FUNCTION_BLOCK UA_UnitMux (* Serialises OPC UA method calls onto command events and routes the accept/reject answer back to the calling method's RSP *)
  (* Standard: 61499-2 *)
  (* Version 2.0, 2026-09-27, Project contributors, Filling cell reference model *)
  PACKAGE fillingcell;
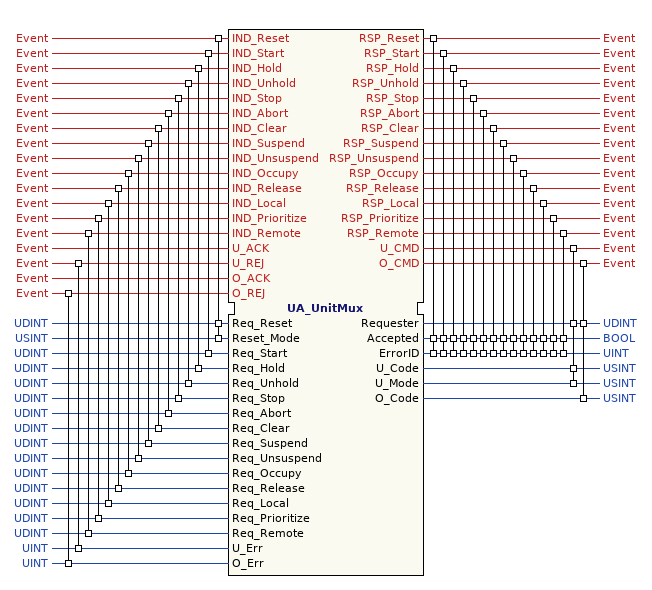
  EVENT_INPUT
    IND_Reset WITH Req_Reset, Reset_Mode;
    IND_Start WITH Req_Start;
    IND_Hold WITH Req_Hold;
    IND_Unhold WITH Req_Unhold;
    IND_Stop WITH Req_Stop;
    IND_Abort WITH Req_Abort;
    IND_Clear WITH Req_Clear;
    IND_Suspend WITH Req_Suspend;
    IND_Unsuspend WITH Req_Unsuspend;
    IND_Occupy WITH Req_Occupy;
    IND_Release WITH Req_Release;
    IND_Local WITH Req_Local;
    IND_Prioritize WITH Req_Prioritize;
    IND_Remote WITH Req_Remote;
    U_ACK;
    U_REJ WITH U_Err;
    O_ACK;
    O_REJ WITH O_Err;
  END_EVENT
  EVENT_OUTPUT
    RSP_Reset WITH Accepted, ErrorID;
    RSP_Start WITH Accepted, ErrorID;
    RSP_Hold WITH Accepted, ErrorID;
    RSP_Unhold WITH Accepted, ErrorID;
    RSP_Stop WITH Accepted, ErrorID;
    RSP_Abort WITH Accepted, ErrorID;
    RSP_Clear WITH Accepted, ErrorID;
    RSP_Suspend WITH Accepted, ErrorID;
    RSP_Unsuspend WITH Accepted, ErrorID;
    RSP_Occupy WITH Accepted, ErrorID;
    RSP_Release WITH Accepted, ErrorID;
    RSP_Local WITH Accepted, ErrorID;
    RSP_Prioritize WITH Accepted, ErrorID;
    RSP_Remote WITH Accepted, ErrorID;
    U_CMD WITH Requester, U_Code, U_Mode;
    O_CMD WITH Requester, O_Code;
  END_EVENT
  VAR_INPUT
    Req_Reset : UDINT;
    Reset_Mode : USINT;
    Req_Start : UDINT;
    Req_Hold : UDINT;
    Req_Unhold : UDINT;
    Req_Stop : UDINT;
    Req_Abort : UDINT;
    Req_Clear : UDINT;
    Req_Suspend : UDINT;
    Req_Unsuspend : UDINT;
    Req_Occupy : UDINT;
    Req_Release : UDINT;
    Req_Local : UDINT;
    Req_Prioritize : UDINT;
    Req_Remote : UDINT;
    U_Err : UINT := 5;
    O_Err : UINT := 5;
  END_VAR
  VAR_OUTPUT
    Requester : UDINT;
    Accepted : BOOL;
    ErrorID : UINT;
    U_Code : USINT;
    U_Mode : USINT;
    O_Code : USINT;
  END_VAR
  VAR
    Pending : USINT;
  END_VAR
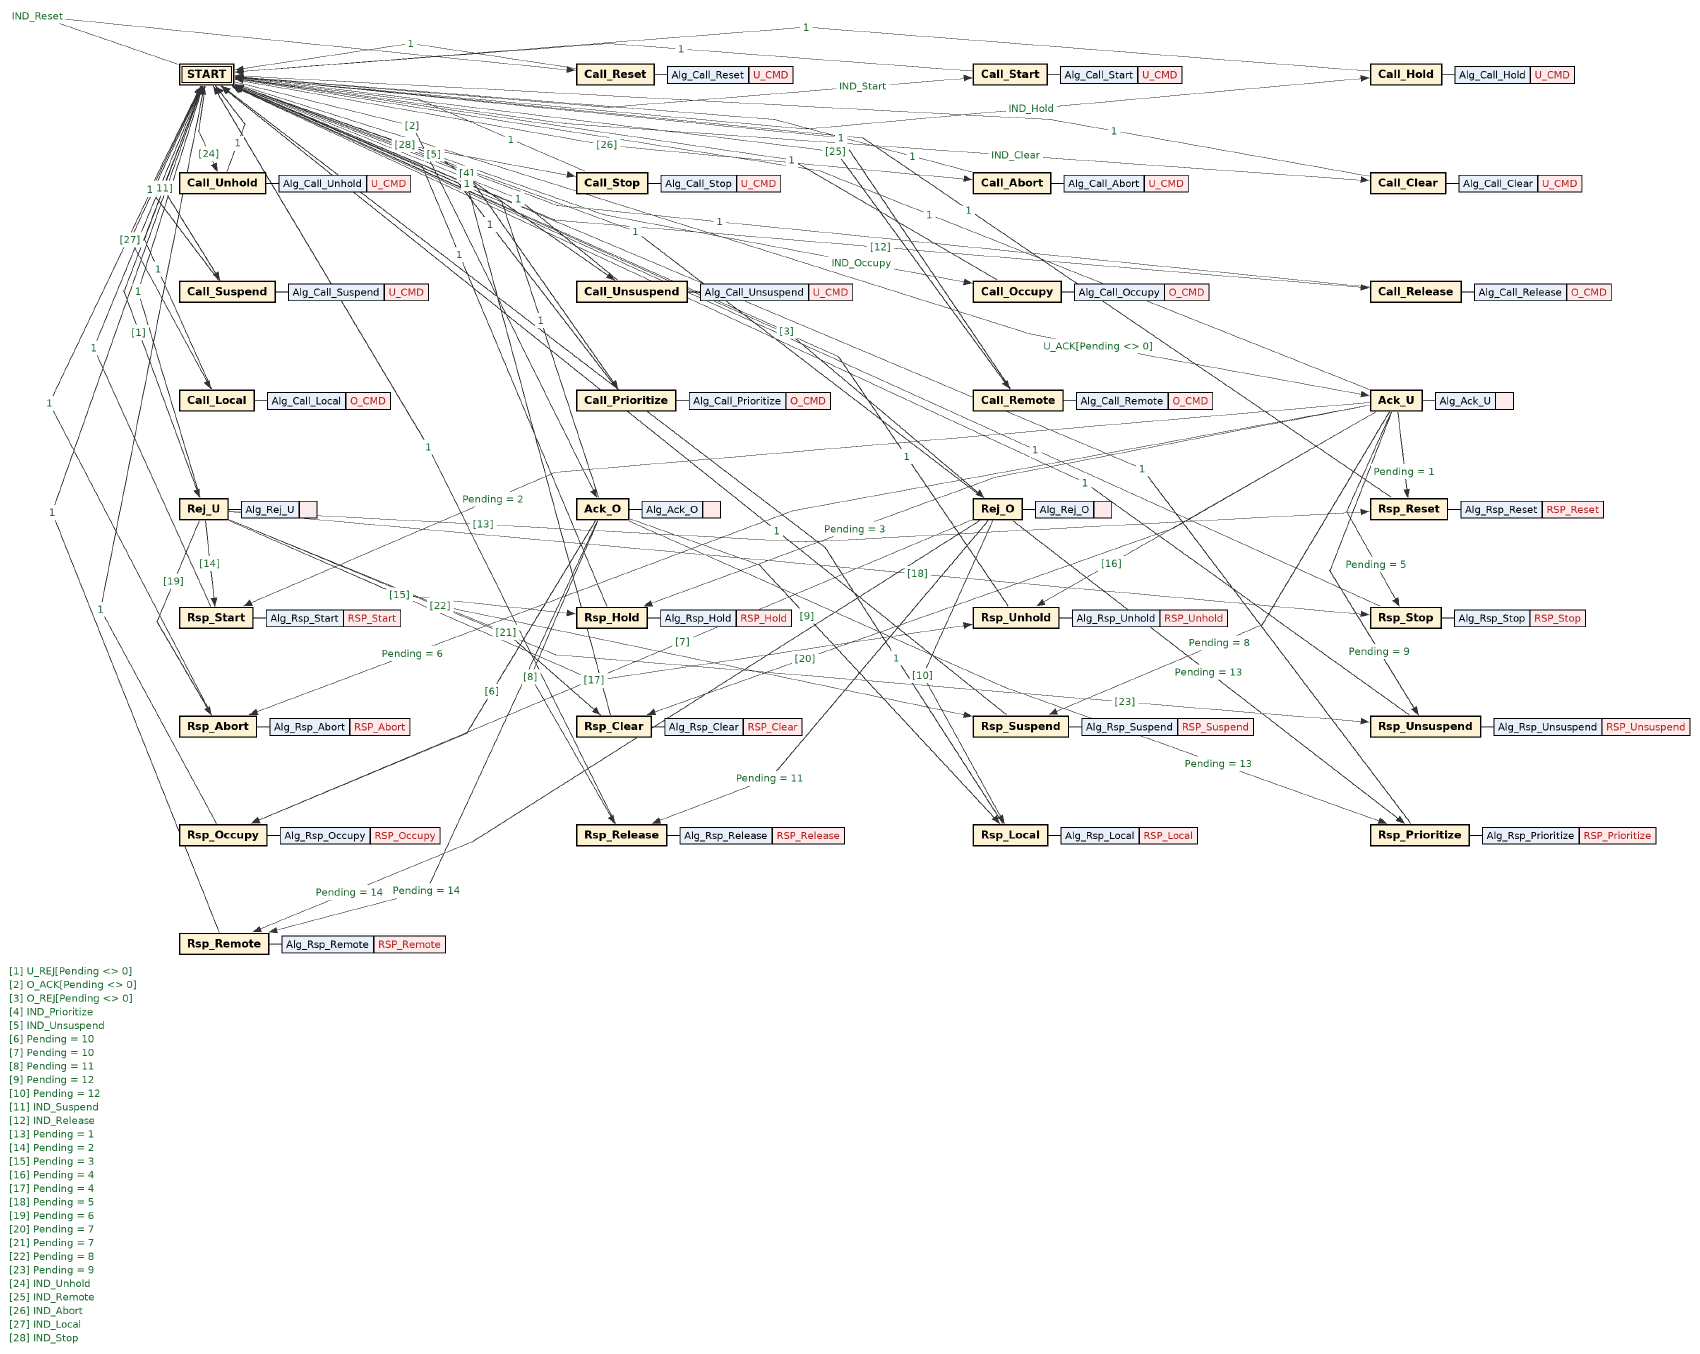
  EC_STATES
    START;
    Call_Reset : Alg_Call_Reset -> U_CMD;
    Call_Start : Alg_Call_Start -> U_CMD;
    Call_Hold : Alg_Call_Hold -> U_CMD;
    Call_Unhold : Alg_Call_Unhold -> U_CMD;
    Call_Stop : Alg_Call_Stop -> U_CMD;
    Call_Abort : Alg_Call_Abort -> U_CMD;
    Call_Clear : Alg_Call_Clear -> U_CMD;
    Call_Suspend : Alg_Call_Suspend -> U_CMD;
    Call_Unsuspend : Alg_Call_Unsuspend -> U_CMD;
    Call_Occupy : Alg_Call_Occupy -> O_CMD;
    Call_Release : Alg_Call_Release -> O_CMD;
    Call_Local : Alg_Call_Local -> O_CMD;
    Call_Prioritize : Alg_Call_Prioritize -> O_CMD;
    Call_Remote : Alg_Call_Remote -> O_CMD;
    Ack_U : Alg_Ack_U;
    Rej_U : Alg_Rej_U;
    Ack_O : Alg_Ack_O;
    Rej_O : Alg_Rej_O;
    Rsp_Reset : Alg_Rsp_Reset -> RSP_Reset;
    Rsp_Start : Alg_Rsp_Start -> RSP_Start;
    Rsp_Hold : Alg_Rsp_Hold -> RSP_Hold;
    Rsp_Unhold : Alg_Rsp_Unhold -> RSP_Unhold;
    Rsp_Stop : Alg_Rsp_Stop -> RSP_Stop;
    Rsp_Abort : Alg_Rsp_Abort -> RSP_Abort;
    Rsp_Clear : Alg_Rsp_Clear -> RSP_Clear;
    Rsp_Suspend : Alg_Rsp_Suspend -> RSP_Suspend;
    Rsp_Unsuspend : Alg_Rsp_Unsuspend -> RSP_Unsuspend;
    Rsp_Occupy : Alg_Rsp_Occupy -> RSP_Occupy;
    Rsp_Release : Alg_Rsp_Release -> RSP_Release;
    Rsp_Local : Alg_Rsp_Local -> RSP_Local;
    Rsp_Prioritize : Alg_Rsp_Prioritize -> RSP_Prioritize;
    Rsp_Remote : Alg_Rsp_Remote -> RSP_Remote;
  END_STATES
  EC_TRANSITIONS
    START TO Call_Reset := IND_Reset;
    Call_Reset TO START := 1;
    START TO Call_Start := IND_Start;
    Call_Start TO START := 1;
    START TO Call_Hold := IND_Hold;
    Call_Hold TO START := 1;
    START TO Call_Unhold := IND_Unhold;
    Call_Unhold TO START := 1;
    START TO Call_Stop := IND_Stop;
    Call_Stop TO START := 1;
    START TO Call_Abort := IND_Abort;
    Call_Abort TO START := 1;
    START TO Call_Clear := IND_Clear;
    Call_Clear TO START := 1;
    START TO Call_Suspend := IND_Suspend;
    Call_Suspend TO START := 1;
    START TO Call_Unsuspend := IND_Unsuspend;
    Call_Unsuspend TO START := 1;
    START TO Call_Occupy := IND_Occupy;
    Call_Occupy TO START := 1;
    START TO Call_Release := IND_Release;
    Call_Release TO START := 1;
    START TO Call_Local := IND_Local;
    Call_Local TO START := 1;
    START TO Call_Prioritize := IND_Prioritize;
    Call_Prioritize TO START := 1;
    START TO Call_Remote := IND_Remote;
    Call_Remote TO START := 1;
    START TO Ack_U := U_ACK[Pending <> 0];
    START TO Rej_U := U_REJ[Pending <> 0];
    START TO Ack_O := O_ACK[Pending <> 0];
    START TO Rej_O := O_REJ[Pending <> 0];
    Ack_U TO Rsp_Reset := Pending = 1;
    Rej_U TO Rsp_Reset := Pending = 1;
    Rsp_Reset TO START := 1;
    Ack_U TO Rsp_Start := Pending = 2;
    Rej_U TO Rsp_Start := Pending = 2;
    Rsp_Start TO START := 1;
    Ack_U TO Rsp_Hold := Pending = 3;
    Rej_U TO Rsp_Hold := Pending = 3;
    Rsp_Hold TO START := 1;
    Ack_U TO Rsp_Unhold := Pending = 4;
    Rej_U TO Rsp_Unhold := Pending = 4;
    Rsp_Unhold TO START := 1;
    Ack_U TO Rsp_Stop := Pending = 5;
    Rej_U TO Rsp_Stop := Pending = 5;
    Rsp_Stop TO START := 1;
    Ack_U TO Rsp_Abort := Pending = 6;
    Rej_U TO Rsp_Abort := Pending = 6;
    Rsp_Abort TO START := 1;
    Ack_U TO Rsp_Clear := Pending = 7;
    Rej_U TO Rsp_Clear := Pending = 7;
    Rsp_Clear TO START := 1;
    Ack_U TO Rsp_Suspend := Pending = 8;
    Rej_U TO Rsp_Suspend := Pending = 8;
    Rsp_Suspend TO START := 1;
    Ack_U TO Rsp_Unsuspend := Pending = 9;
    Rej_U TO Rsp_Unsuspend := Pending = 9;
    Rsp_Unsuspend TO START := 1;
    Ack_O TO Rsp_Occupy := Pending = 10;
    Rej_O TO Rsp_Occupy := Pending = 10;
    Rsp_Occupy TO START := 1;
    Ack_O TO Rsp_Release := Pending = 11;
    Rej_O TO Rsp_Release := Pending = 11;
    Rsp_Release TO START := 1;
    Ack_O TO Rsp_Local := Pending = 12;
    Rej_O TO Rsp_Local := Pending = 12;
    Rsp_Local TO START := 1;
    Ack_O TO Rsp_Prioritize := Pending = 13;
    Rej_O TO Rsp_Prioritize := Pending = 13;
    Rsp_Prioritize TO START := 1;
    Ack_O TO Rsp_Remote := Pending = 14;
    Rej_O TO Rsp_Remote := Pending = 14;
    Rsp_Remote TO START := 1;
    Ack_U TO START := 1;
    Rej_U TO START := 1;
    Ack_O TO START := 1;
    Rej_O TO START := 1;
  END_TRANSITIONS
  ALGORITHM Alg_Call_Reset IN ST:
Requester := Req_Reset;
U_Code := 1;
U_Mode := Reset_Mode;
Pending := 1;
  END_ALGORITHM
  ALGORITHM Alg_Call_Start IN ST:
Requester := Req_Start;
U_Code := 2;
Pending := 2;
  END_ALGORITHM
  ALGORITHM Alg_Call_Hold IN ST:
Requester := Req_Hold;
U_Code := 3;
Pending := 3;
  END_ALGORITHM
  ALGORITHM Alg_Call_Unhold IN ST:
Requester := Req_Unhold;
U_Code := 4;
Pending := 4;
  END_ALGORITHM
  ALGORITHM Alg_Call_Stop IN ST:
Requester := Req_Stop;
U_Code := 5;
Pending := 5;
  END_ALGORITHM
  ALGORITHM Alg_Call_Abort IN ST:
Requester := Req_Abort;
U_Code := 6;
Pending := 6;
  END_ALGORITHM
  ALGORITHM Alg_Call_Clear IN ST:
Requester := Req_Clear;
U_Code := 7;
Pending := 7;
  END_ALGORITHM
  ALGORITHM Alg_Call_Suspend IN ST:
Requester := Req_Suspend;
U_Code := 8;
Pending := 8;
  END_ALGORITHM
  ALGORITHM Alg_Call_Unsuspend IN ST:
Requester := Req_Unsuspend;
U_Code := 9;
Pending := 9;
  END_ALGORITHM
  ALGORITHM Alg_Call_Occupy IN ST:
Requester := Req_Occupy;
O_Code := 1;
Pending := 10;
  END_ALGORITHM
  ALGORITHM Alg_Call_Release IN ST:
Requester := Req_Release;
O_Code := 2;
Pending := 11;
  END_ALGORITHM
  ALGORITHM Alg_Call_Local IN ST:
Requester := Req_Local;
O_Code := 3;
Pending := 12;
  END_ALGORITHM
  ALGORITHM Alg_Call_Prioritize IN ST:
Requester := Req_Prioritize;
O_Code := 4;
Pending := 13;
  END_ALGORITHM
  ALGORITHM Alg_Call_Remote IN ST:
Requester := Req_Remote;
O_Code := 5;
Pending := 14;
  END_ALGORITHM
  ALGORITHM Alg_Ack_U IN ST:
Accepted := TRUE;
ErrorID := 0;
  END_ALGORITHM
  ALGORITHM Alg_Rej_U IN ST:
Accepted := FALSE;
ErrorID := U_Err;
  END_ALGORITHM
  ALGORITHM Alg_Ack_O IN ST:
Accepted := TRUE;
ErrorID := 0;
  END_ALGORITHM
  ALGORITHM Alg_Rej_O IN ST:
Accepted := FALSE;
ErrorID := O_Err;
  END_ALGORITHM
  ALGORITHM Alg_Rsp_Reset IN ST:
Pending := 0;
  END_ALGORITHM
  ALGORITHM Alg_Rsp_Start IN ST:
Pending := 0;
  END_ALGORITHM
  ALGORITHM Alg_Rsp_Hold IN ST:
Pending := 0;
  END_ALGORITHM
  ALGORITHM Alg_Rsp_Unhold IN ST:
Pending := 0;
  END_ALGORITHM
  ALGORITHM Alg_Rsp_Stop IN ST:
Pending := 0;
  END_ALGORITHM
  ALGORITHM Alg_Rsp_Abort IN ST:
Pending := 0;
  END_ALGORITHM
  ALGORITHM Alg_Rsp_Clear IN ST:
Pending := 0;
  END_ALGORITHM
  ALGORITHM Alg_Rsp_Suspend IN ST:
Pending := 0;
  END_ALGORITHM
  ALGORITHM Alg_Rsp_Unsuspend IN ST:
Pending := 0;
  END_ALGORITHM
  ALGORITHM Alg_Rsp_Occupy IN ST:
Pending := 0;
  END_ALGORITHM
  ALGORITHM Alg_Rsp_Release IN ST:
Pending := 0;
  END_ALGORITHM
  ALGORITHM Alg_Rsp_Local IN ST:
Pending := 0;
  END_ALGORITHM
  ALGORITHM Alg_Rsp_Prioritize IN ST:
Pending := 0;
  END_ALGORITHM
  ALGORITHM Alg_Rsp_Remote IN ST:
Pending := 0;
  END_ALGORITHM
END_FUNCTION_BLOCK
